(* IEC 61131-3 sources: TSA-FMICS22/ahorn/test/lib_pass/file/tac, 4 files *)

(* ---- boolean_assignments.st ---- *)
PROGRAM P
VAR
    x : INT;
    y : INT;
    b1 : BOOL;
    b2 : BOOL;
    b3 : BOOL;
END_VAR
    b1 := x + x < y;
    b2 := x + x = y;
    b3 := x + x > y;
END_PROGRAM

(* ---- consecutive_assignments.st ---- *)
PROGRAM P
VAR
    a : INT;
    b : INT;
    c : INT;
    d : INT;
END_VAR
    a := b + c + d;
    b := a * a + b * b;
END_PROGRAM

(* ---- parts_of_antivalent.st ---- *)
PROGRAM P
VAR_INPUT
    Activate       : BOOL := FALSE;
END_VAR
VAR
    Ready          : BOOL := FALSE;
    S_TwoHandOut   : BOOL := FALSE;
    DiagCode       : WORD := 16#0;
END_VAR
    IF NOT Activate THEN
        DiagCode := 16#0000;
    ELSE
     CASE DiagCode OF
     16#0000:
         IF Activate THEN
              DiagCode := 16#8001;
         END_IF;
     END_CASE;
    END_IF;

    CASE DiagCode OF
    16#0000:
        Ready := FALSE;
        S_TwoHandOut := FALSE;
    16#8000:
        Ready := TRUE;
        S_TwoHandOut := TRUE;
    16#8001:
        Ready := TRUE;
        S_TwoHandOut := FALSE;
    END_CASE;
END_PROGRAM

(* ---- preserve_operand_order.st ---- *)
PROGRAM P
VAR
    a : INT;
    b : INT;
END_VAR
    a := 5 + 2 * b;
END_PROGRAM
